// TIA Portal V20 export
TYPE "IO_AO"
   STRUCT
      OUT : Struct
         ValueOut : Real;
      END_STRUCT;
   END_STRUCT;
END_TYPE
